// TwinCAT 3 PLC project PLC
// ProgramVersion: 3.1.4026.20
// libraries:
//   Tc2_MC2, * (Beckhoff Automation GmbH)
//   Tc2_Standard, * (Beckhoff Automation GmbH)
//   Tc2_System, * (Beckhoff Automation GmbH)
// project tree:
//   DUTs/ EAnlageGes.TcDUT, EAnlagenStatus.TcDUT, EFoerderband.TcDUT, ETransport.TcDUT
//   GVLs/ IFC_HW.TcGVL
//   / PlcTask.TcTTO
//   POUs/ FB_Abfuellmodul.TcPOU, FB_DigitalInput.TcPOU, FB_Dispenser.TcPOU, MAIN.TcPOU, F_SensStationMonitor.TcPOU
//   POUs/Fehlerbehandlung/ FB_TimeOutError.TcPOU
//   POUs/HardwareEbene/ FB_StatusLight.TcPOU, FB_CNV.TcPOU, FB_RCtrl.TcPOU, FB_Transport.TcPOU
//   POUs/ProzessEbene/ FB_Vereinzelung.TcPOU (not stored)
// (motion and I/O tree: see PLC project tempmodel)
// real-time tasks:
//   TASK PlcTask: cycle T#10ms, priority 21, ADS port 350
//   TASK PlcTask1: cycle T#10ms, priority 22, ADS port 351
//   TASK PlcTask2: cycle T#10ms, priority 20, ADS port 352
// variable links:
//   LF_System_PLC/LF_System_PLC Instance <-> PLC/PLC Instance
//     PlcTask Inputs/MAIN.bIn_LedGreen <-> PlcTask Outputs/IFC_HW.bAmpelGrun
//     PlcTask Inputs/MAIN.bIn_LedRot <-> PlcTask Outputs/IFC_HW.bAmpelRot
//     PlcTask Inputs/MAIN.bIn_LedYellow <-> PlcTask Outputs/IFC_HW.bAmpelGelb
//     PlcTask Inputs/MAIN.bIn_Schleuse1_L1 <-> PlcTask Outputs/IFC_HW.bR1AKT1
//     PlcTask Inputs/MAIN.bIn_Schleuse1_L2 <-> PlcTask Outputs/IFC_HW.bR2AKT1
//     PlcTask Inputs/MAIN.bIn_Schleuse2_L1 <-> PlcTask Outputs/IFC_HW.bR1AKT2
//     PlcTask Inputs/MAIN.bIn_Schleuse2_L2 <-> PlcTask Outputs/IFC_HW.bR2AKT2
//     PlcTask Outputs/MAIN.bEnable <-> PlcTask Inputs/IFC_HW.bEnable
//     PlcTask Outputs/MAIN.bExecute <-> PlcTask Inputs/IFC_HW.bExecute
//     PlcTask Outputs/MAIN.bOut_VereinzelungNS1 <-> PlcTask Inputs/IFC_HW.bEinzelSens3
//     PlcTask Outputs/MAIN.bOut_VereinzelungNS2 <-> PlcTask Inputs/IFC_HW.bEinzelSens2
//     PlcTask Outputs/MAIN.bOut_VereinzelungNS3 <-> PlcTask Inputs/IFC_HW.bEinzelSens1
//   PLC/PLC Instance <-> NC-Task 1 SAF/Axes/BandAchse
//     PlcTask Inputs/IFC_HW.ax_BandMotor.NcToPlc <-> Outputs/ToPlc
//     PlcTask Outputs/IFC_HW.ax_BandMotor.PlcToNc <-> Inputs/FromPlc

CONFIGURATION PLC
    RESOURCE PLC ON TwinCAT3
        TASK PlcTask(INTERVAL := T#10ms, PRIORITY := 20);
        PROGRAM MAIN WITH PlcTask : MAIN;
    END_RESOURCE
END_CONFIGURATION

// ---- DUTs/EAnlageGes.TcDUT
{attribute 'qualified_only'}
{attribute 'strict'}
{attribute 'to_string'}
TYPE EFoerderband :
(
	Off:=0,
	Init := 1,
	Ready := 2,
	Production := 3,
	Done := 4	
);
END_TYPE

// ---- DUTs/EAnlagenStatus.TcDUT
{attribute 'qualified_only'}
{attribute 'strict'}
{attribute 'to_string'}
TYPE EAnlagenStatus:
(
	OFF := 0,
	StateInitOpen := 10,
	StateInitClose := 11,
	StateReady := 20,
	StateProductionOpen := 30,
	StateProductionClose := 31,
	StateDone := 40	
);
END_TYPE

// ---- DUTs/EFoerderband.TcDUT
{attribute 'qualified_only'}
{attribute 'strict'}
{attribute 'to_string'}
TYPE EFoerderband :
(
	Off:=0,
	init := 1,
	ErrorState := 99,
	Resolve := 100,
	Ready := 2,
	CNV_on := 3,
	CNV:aus := 4,
	Done := 5
	
);
END_TYPE

// ---- DUTs/ETransport.TcDUT
{attribute 'qualified_only'}
{attribute 'strict'}
{attribute 'to_string'}
TYPE ETransport :
(
	Off:=0,
	Init := 1,
	Ready := 2,
	Production := 3,
	Producing := 4,
	Done := 5
);
END_TYPE

// ---- GVLs/IFC_HW.TcGVL
// In dieser GVL werden alle Variablen deklariert die auf die realen Klemmen zugreifen
VAR_GLOBAL
	
	// Allgemeine Variablen fur MAIN und HMI
		bEnable		AT%I*	: BOOL;			// Enable Factory (HMI Production Umgebung)
		bExecute	AT%I*	: BOOL;			// Startsignal	(Start Knopf Konsole)
		bStop				: BOOL;			// Stop Variable (interne Variable um FB's zu stoppen)
		bReset				: BOOL;			// Reset Variable
		
	// Station Statusampel	
		bAmpelRot 	AT%Q* 	: BOOL;			// Signal-LED Rot
		bAmpelGelb 	AT%Q* 	: BOOL;			// Signal-LED Gelb
		bAmpelGrun 	AT%Q* 	: BOOL;			// Signal-LED Grun
			
	// Station Vereinzelung
		bEinzelSens1 	AT%I*	: BOOL;					// Separation Sensor 1 (Kammer)
		bEinzelSens2 	AT%I*	: BOOL;					// Separation Sensor 2 (Rohr)
		bEinzelSens3 	AT%I*	: BOOL;					// Separation Sensor 3 (Flasche auf Kopf)
		bR1AKT1 		AT%Q* 	: BOOL := FALSE;		// Relais 1 Aktor 1 (Schleuse Oben öffnen)
		bR2AKT1 		AT%Q* 	: BOOL := TRUE; 		// Relais 2 Aktor 1 (Schleuse Oben schließen)
		bR1AKT2 		AT%Q* 	: BOOL := FALSE;		// Relais 1 Aktor 2 (Schleuse Unten öffne)
		bR2AKT2 		AT%Q* 	: BOOL := TRUE;			// Relais 2 Aktor 2	(Schleuse Unten schließen)
	
	// Station Forderband
		bBandSens1 	AT %I*	: BOOL;		// Forderband Sensor 1 (Extruder 1)
		bBandSens2	AT %I*	: BOOL;		// Forderband Sensor 2 (Extruder 2)
		bBandSens3 	AT %I*	: BOOL;		// Forderband Sensor 3 (Extruder 3)
		bBandSens4 	AT %I*	: BOOL;		// Forderband Sensor 4 (Übergabe Roboter)
		bBandHub1 	AT %Q*	: BOOL;		// Forderband Hubmagnet 1 (Schleuse Extruder 1)
		bBandHub2 	AT %Q*	: BOOL;		// Forderband Hubmagnet 1 (Schleuse Extruder 2)
		bBandHub3 	AT %Q*	: BOOL;		// Forderband Hubmagnet 1 (Schleuse Extruder 3)
		
		ax_Extruder1 	: AXIS_REF;		// Forderband NC-Achse Extruder 1
		ax_Extruder2 	: AXIS_REF;		// Forderband NC-Achse Extruder 2
		ax_Extruder3 	: AXIS_REF;		// Forderband NC-Achse Extruder 3
		ax_BandMotor 	: AXIS_REF;		// Forderband NC-Achse Band
		
		iBandFullmenge1		: INT := 1;	// in Gramm (Soll Füllmenge Extruder 1)
		iBandFullmenge2		: INT := 1;	// in Gramm (Soll Füllmenge Extruder 2)
		iBandFullmenge3		: INT := 1;	// in Gramm (Soll Füllmenge Extruder 3)
		
	//Füllstandsüberwachung
		iFillSens1 AT%I*	: UINT;		// Füllstandssensor im Granulatspeicher 1
		iFillSens2 AT%I*	: UINT;		// Füllstandssensor im Granulatspeicher 2
		iFillSens3 AT%I*	: UINT;		// Füllstandssensor im Granulatspeicher 3
		
		rFillLevelPercent1	: REAL;		// Füllstand im Granulatspeicher 1 in %
		rFillLevelGramm1	: REAL;		// Füllstand im Granulatspeicher 1 in g
		rFillLevelPercent2	: REAL;		// Füllstand im Granulatspeicher 2 in %
		rFillLevelGramm2	: REAL;		// Füllstand im Granulatspeicher 2 in g
		rFillLevelPercent3	: REAL;		// Füllstand im Granulatspeicher 3 in %
		rFillLevelGramm3	: REAL;		// Füllstand im Granulatspeicher 3 in g
		
		rMaxFillLevel 		: REAL := 375;	// Kalibrierter Füllstand für 10% * 10
		
	// Station Waage
		sWaageNachricht		: STRING;	// Nachricht von Wagezelle (fur virtuelle Inbetriebnahme notig)
		bWaageNull			: BOOL;		// TARA Waage (Waage auf Null setzen)
		iWaageMesswert		: INT;		// Messwert der Waage
		
	// Station Behalteridentifikation
		bIdSensorTrager		: BOOL;		// Sensor bei Erkennung eines Datentrager
		sIdNachricht		: STRING;	// Nachricht von RFID-System (fur virtuelle Inbetriebnahme notig)
		sSeriennummer		: STRING;	// Seriennummer RFID-Tag
		
	//Temperierstation
		bVentilator1 	AT %Q*	: BOOL;		// Ventilator 1
		bVentilator2 	AT %Q*	: BOOL;		// Ventilator 2
		bVentilator3 	AT %Q*	: BOOL;		// Ventilator 3
		
		iTempSens1 		AT%I*	: UINT;		// Temperatursensor 1
		iTempSens2 		AT%I*	: UINT;		// Temperatursensor 2
		iHeizpatrone 	AT%Q*	: UINT;		// Heizpatronen
		
		iMaxTemp				: UINT := 5500;		// in °C * 100
		
	// Station Manipulator
		bManEndXmin 		AT%I* 	: BOOL := TRUE;		// Manipulator min Endschalter Achse x
		bManEndYmin 		AT%I* 	: BOOL := TRUE;		// Manipulator min Endschalter Achse y
		bManEndZmin 		AT%I* 	: BOOL := TRUE;		// Manipulator min Endschalter Achse z
		bManEndGmin 		AT%I* 	: BOOL := TRUE;		// Manipulator min Endschalter Achse Gripper
		bManEndXmax 		AT%I* 	: BOOL := TRUE;		// Manipulator max Endschalter Achse x
		bManEndYmax 		AT%I* 	: BOOL := TRUE;		// Manipulator max Endschalter Achse y
		bManEndZmax 		AT%I* 	: BOOL := TRUE;		// Manipulator max Endschalter Achse z
		bManEndGmax 		AT%I* 	: BOOL := TRUE;		// Manipulator max Endschalter Achse Gripper
		bManBrakeZ			AT%Q*	: BOOL := FALSE;	// Bremse Achse z
		
		ax_ManX			: AXIS_REF;			// Manipulator NC-Achse x
		ax_ManY			: AXIS_REF;			// Manipulator NC-Achse y
		ax_ManZ			: AXIS_REF;			// Manipulator NC-Achse z
		ax_ManG			: AXIS_REF; 		// Manipulator NC-Achse Gripper
		
		bGripperClosed		AT%Q*	: BOOL; 			// signal if gripper is closed ONLY USED IN SIM
END_VAR

// ---- POUs/MAIN.TcPOU
PROGRAM MAIN
VAR
	bRed : BOOL;
	bGreen : BOOL;
	bYellow : BOOL;
	
	// FB_Vereinzelung_In:
	bSens1 : BOOL;
	bSens2 : BOOL;
	bSens3 : BOOL;
	bEnable : BOOL;
	bExecute : BOOL;
	
	// FB_Vereinzelung_OUT:
	bGate1 : BOOL;
	bGate2 : BOOL;
	
	fbVereinzelung : FB_Vereinzelung;
	fbRctrl : fb_RCtrl;	
	fbBlink : FB_StatusLight;
	fbCNV : FB_CNV;
	fbEndXmin : FB_DigitalInput(TRUE);
	fbAbfuellmodul : FB_Abfuellmodul;
	
	eStatus : EAnlagenStatus;
	nDoneCounter : INT;
	bError : BOOL;
	ErrorID : DWORD;
	bReset : BOOL;
	
	
	
END_VAR

fbCNV(
	bEnable:= ifc_hw.bEnable, 
	bExecute:= ifc_hw.bExecute, 
	bHalt:= ifc_hw.bBandSens1, 
	rVel:= 50, 
	ax:= ifc_hw.ax_BandMotor);
	
fbEndXmin (bsensSignal := Ifc_HW.bManEndXmin , bSensLogic =>);

IF fbEndXmin.bSensLogic THEN
	//Achse darf nicht in negative Richtung fahren
END_IF
	
fbVereinzelung(
	bSens1 := IFC_HW.bEinzelSens1,
	bSens2 := IFC_HW.bEinzelSens2,
	bSens3 := IFC_HW.bEinzelSens3,
	bEnable := IFC_HW.bEnable,
	bExecute := IFC_HW.bExecute,
	bGate1 => bGate1,
	bGate2 => bGate2,
	eStatus => eStatus,
	nDoneCounter => nDoneCounter);
	
bGate1 := fbVereinzelung.bGate1;
bGate2 := fbVereinzelung.bGate2;

fbRctrl(
	bGate1 := bGate1,
	bGate2 := bGate2,
	bGate1Auf=> IFC_HW.bR1AKT1, 
	bGate1Zu=> IFC_HW.bR2AKT1, 
	bGate2Auf=> IFC_HW.bR1AKT2, 
	bGate2Zu=> IFC_HW.bR2AKT2);

fbAbfuellmodul(
	bEnable:= , 
	bExecute:= , 
	eState=> , 
	bError=> bError, 
	ErrorID=> ErrorID);

fbBlink(eStatus:= eStatus, bRed=> IFC_HW.bAmpelRot, bGreen=> IFC_HW.bAmpelGrun, bYellow=> IFC_HW.bAmpelGelb);

IF bError AND (ErrorID = 9001 OR ErrorID = 9003) THEN
	ifc_HW.bstop := TRUE;
END_IF

ifc_HW.bReset := bReset;
	
IF breset AND NOT bError THEN
	ifc_HW.bStop := FALSE;
	breset := FALSE;
END_IF
(*
//OUT
IFC_HW.bAmpelRot := bRed;
IFC_HW.bAmpelGrun := bGreen;
IFC_HW.bAmpelGelb := bYellow;

IFC_HW.bR1AKT1 := bGate1Auf; //Schleuse oben öffnen
IFC_HW.bR2AKT1 := bGate1Zu;
IFC_HW.bR1AKT2 := bGate2Auf;
IFC_HW.bR2AKT2 := bGate2Zu;

//IN
bSens1 := IFC_HW.bEinzelSens1;
bSens2 := IFC_HW.bEinzelSens1;
bSens3 := IFC_HW.bEinzelSens3;

bEnable := IFC_HW.bEnable;
bExecute := IFC_HW.bExecute;
*)

END_PROGRAM

// ---- POUs/HardwareEbene/FB_RCtrl.TcPOU
FUNCTION_BLOCK FB_RCtrl
VAR_INPUT
	bGate1 : BOOL;
	bGate2 : BOOL;
	
END_VAR
VAR_OUTPUT
	bGate1Auf : BOOL;
	bGate1Zu : BOOL;
	bGate2Auf : BOOL;
	bGate2Zu : BOOL;
END_VAR
VAR
END_VAR

IF bGate1 THEN
	bGate1Auf := TRUE;
	bGate1Zu := FALSE;
	bGate2Auf := FALSE;
	bGate2Zu := TRUE;

ELSIF bGate2 THEN
	bGate1Auf := FALSE;
	bGate1Zu := TRUE;
	bGate2Auf := TRUE;
	bGate2Zu := FALSE;

ELSIF NOT bGate1 THEN
	bGate1Auf := FALSE;
	bGate1Zu := TRUE;

ELSIF NOT bGate2 THEN
	bGate2Auf := FALSE;
	bGate2Zu := TRUE;
	
END_IF

END_FUNCTION_BLOCK

// ---- POUs/HardwareEbene/FB_StatusLight.TcPOU
FUNCTION_BLOCK FB_StatusLight
VAR_INPUT
	eStatus : EAnlagenStatus;
	//bEnable : BOOL; //für stop status
	
END_VAR
VAR_OUTPUT
	bRed : BOOL;
	bGreen : BOOL;
	bYellow : BOOL;
	
END_VAR
VAR
	bblinkEnable : BOOL := FALSE;
	bblinkNow : BOOL := FALSE;
	
	bblinkRED : BOOL := FALSE;
	bblinkGreen : BOOL := FALSE;
	bblinkYellow : BOOL := FALSE;
	
	fbTON : TON;
	fbTP : TP;

END_VAR

bblinkEnable := FALSE;
bblinkNow := FALSE;
	
bblinkRED := FALSE;
bblinkGreen := FALSE;
bblinkYellow := FALSE;

bRed    := FALSE;
bGreen  := FALSE;
bYellow := FALSE;

CASE eStatus OF
	EAnlagenStatus.OFF:
		bRed := TRUE;
		bblinkEnable := FALSE;
		
	EAnlagenStatus.StateInitOpen, EAnlagenStatus.StateInitClose:	//Init
		bblinkEnable := TRUE;
		bblinkGreen := TRUE;
		bblinkRed := FALSE;
		bblinkYellow := FALSE;
		
	EAnlagenStatus.StateProductionOpen, EAnlagenStatus.StateProductionClose: //Production
		bblinkEnable := FALSE;
		bGreen := TRUE;
		
	EAnlagenStatus.StateReady: //Ready
		bblinkEnable := TRUE;
		bblinkGreen := TRUE;
		bblinkyellow := TRUE;
	
	EAnlagenStatus.StateDone: //Done
		bblinkEnable := FALSE;
		bGreen := TRUE;
		bYellow := TRUE;
	
	
END_CASE

fbTON(IN:=bblinkEnable AND NOT fbTon.Q , PT:= T#1S , Q=> , ET=> );
fbTP(IN:= fbTon.Q, PT:= T#500MS , Q=> , ET=> );

bblinkNow := fbTP.Q;

IF bblinkEnable THEN
		
	IF bblinkRed THEN
		bRed := bblinkNow;	
	END_IF
	
	IF bblinkGreen THEN
		bGreen := bblinkNow;
	END_IF
	
	IF bblinkYellow THEN
		bYellow := bblinkNow;
	END_IF
END_IF

END_FUNCTION_BLOCK

// ---- POUs/HardwareEbene/FB_CNV.TcPOU
FUNCTION_BLOCK FB_CNV
VAR_INPUT
	bEnable : BOOL;
	bExecute : BOOL;
	bHalt : BOOL;
	rVel : REAL;
	
	eState : EFoerderband;
END_VAR
VAR_OUTPUT
END_VAR
VAR
	nState : INT :=0;
	mcPower : MC_Power;
	mcReset : MC_Reset;
	mcVelocity : MC_MoveVelocity;
	mcHalt : MC_Halt;
	ErrorID: INT;
	bStop : Bool;
	mcStop: MC_Stop;
END_VAR

VAR_IN_OUT 
	ax : Axis_Ref;
END_VAR

mcHalt(
	Axis:= ax, 
	Execute:= , 
	Deceleration:= , 
	Jerk:= , 
	BufferMode:= , 
	Options:= , 
	Done=> , 
	Busy=> , 
	Active=> , 
	CommandAborted=> , 
	Error=> , 
	ErrorID=> );
	
mcPower(
	Axis:= ax, 
	Enable:= , 
	Enable_Positive:= , 
	Enable_Negative:= , 
	Override:= , 
	BufferMode:= , 
	Options:= , 
	Status=> , 
	Busy=> , 
	Error=> , 
	ErrorID=> );
	
mcReset(
	Axis:= ax, 
	Execute:= , 
	Done=> , 
	Busy=> , 
	Error=> , 
	ErrorID=> );
	
mcVelocity(
	Axis:= ax, 
	Execute:= , 
	Velocity:= rVel, 
	Acceleration:= , 
	Deceleration:= , 
	Jerk:= , 
	Direction:= , 
	BufferMode:= , 
	Options:= , 
	InVelocity=> , 
	Busy=> , 
	Active=> , 
	CommandAborted=> , 
	Error=> , 
	ErrorID=> );

ax.ReadStatus();

bStop := ifc_HW.bStop;
IF bStop THEN
	nState := 80;
END_IF

IF ax.Status.Error THEN 
	nState := 99;
ELSIF NOT bEnable THEN 
	nState := 0;
END_IF

CASE eState OF
	EFoerderband.Off: // OFF
	
		mcReset.Execute := FALSE;
		mcPower.Enable := FALSE;
		mcPower.Enable_Positive := FALSE;
		mcVelocity.Execute := FALSE;
		mcHalt.Execute := FALSE;
		
		
		IF ax.Status.Error THEN 
			nState := 99;
		ELSIF bEnable THEN 
			nState := 1;
		END_IF
	
	EFoerderband.init: //INIT
		
		mcPower.Enable := TRUE;
		mcPower.Enable_Positive := FALSE;
		mcReset.Execute := FALSE;
		mcVelocity.Execute := FALSE;
		mcHalt.Execute := FALSE;
	
		IF mcPower.Status THEN 
			nState :=2;
		END_IF
		
	EFoerderband.Ready: //Ready
		mcPower.Enable := TRUE;
		mcPower.Enable_Positive := FALSE;
		mcReset.Execute := FALSE;
		mcVelocity.Execute := FALSE;
		mcHalt.Execute := FALSE;
		
		IF bExecute THEN 
			nState :=3;
		END_IF
	
	EFoerderband.CNV_on:// CNV an
		mcPower.Enable := TRUE;
		mcPower.Enable_Positive := TRUE;
		mcReset.Execute := FALSE;
		mcVelocity.Execute := TRUE;
		mcHalt.Execute := FALSE;
		
		IF bHalt THEN 
			nState :=4;
		END_IF
	
	EFoerderband.CNV_aus: // CNV aus
		mcPower.Enable := TRUE;
		mcPower.Enable_Positive := TRUE;
		mcReset.Execute := FALSE;
		mcVelocity.Execute := FALSE;
		mcHalt.Execute := TRUE;
		
		IF mcHalt.Done THEN 
			nState :=5;
		END_IF
	
	EFoerderband.Done: // DONE
		mcPower.Enable := TRUE;
		mcPower.Enable_Positive := TRUE;
		mcReset.Execute := FALSE;
		mcVelocity.Execute := FALSE;
		mcHalt.Execute := FALSE;
		
		IF NOT bExecute AND NOT bHalt THEN 
			nState :=2;
		END_IF
	
	EFoerderband.ErrorState: // ERROR 
		mcPower.Enable := FALSE;
		mcPower.Enable_Positive := FALSE;
		mcReset.Execute := FALSE;
		mcVelocity.Execute := FALSE;
		mcHalt.Execute := FALSE;
		
		IF bEnable THEN 
			nState :=100;
		END_IF
	80: //Stop CNV
	mcVelocity.Execute := FALSE;
	mcHalt.Execute := FALSE;
	mcStop.Execute := TRUE;
	
	81: //RE-INIT //noch überarbeiten mit e state und 
	mcVelocity.Execute := FALSE;
	mcHalt.Execute := FALSE;
	mcStop.Execute := FALSE;
	mcReset //auch noch setzen 
	
	
	EFoerderband.Resolve: // Resolve
		mcPower.Enable := TRUE;
		mcPower.Enable_Positive := TRUE;
		mcReset.Execute := FALSE;
		mcVelocity.Execute := FALSE;
		mcHalt.Execute := FALSE;
	
	IF mcReset.Done THEN 
			nState :=1;
		END_IF
END_CASE

END_FUNCTION_BLOCK

// ---- POUs/FB_DigitalInput.TcPOU
FUNCTION_BLOCK FB_DigitalInput
VAR_INPUT
	bSensSignal : BOOL;
END_VAR
VAR_OUTPUT
	bSensLogic : BOOL;
END_VAR
VAR
	_Invert : BOOL := FALSE; //_ damit man weiß ist eine interne variable
END_VAR

IF _Invert THEN
	bSensLogic := NOT bSensSignal;
ELSE
	bSensLogic := bSensSignal;
END_IF

//FB_Init is always available implicitly and it is used primarily for initialization.
//The return value is not evaluated. For a specific influence, you can also declare the
//methods explicitly and provide additional code there with the standard initialization
//code. You can evaluate the return value.
METHOD FB_Init: BOOL
VAR_INPUT
    bInitRetains: BOOL; // TRUE: the retain variables are initialized (reset warm / reset cold)
    bInCopyCode: BOOL;  // TRUE: the instance will be copied to the copy code afterward (online change)   
	Invert : BOOL;
END_VAR
_Invert := Invert;
END_METHOD

END_FUNCTION_BLOCK

// ---- POUs/FB_Abfuellmodul.TcPOU
FUNCTION_BLOCK FB_Abfuellmodul
VAR_INPUT
	bEnable : BOOL;
	bExecute : BOOL;
END_VAR
VAR_OUTPUT
	eState : EAnlageGes;
	bError : BOOL;
	ErrorID : DWORD;
END_VAR
VAR
	fbTransport : FB_Transport;
	fbDispenser : FB_Dispenser;
	nState : INT;
	bStop : BOOL;
END_VAR

fbTransport(
	bSens1:= , 
	bSens2:= , 
	bSens3:= , 
	bSens4:= , 
	bEnabale:= , 
	bExecute:= , 
	nStation:= , 
	eState:= , 
	fSensStationMonitor:= , 
	bHub1=> , 
	bHub2=> , 
	bHub3=> , 
	bError=> bError, 
	ErrorID=> ErrorID);
	
	bStop := ifc_HW.bStop;
	
	IF NOT bEnable THEN
		//noch auszuarbeiten
	END_IF
	
	IF NOT bStop THEN
		CASE nState OF
			//noch auszuarbeiten
		END_CASE
	END_IF

END_FUNCTION_BLOCK

// ---- POUs/HardwareEbene/FB_Transport.TcPOU
FUNCTION_BLOCK FB_Transport
VAR_INPUT
	bSens1 : BOOL;
	bSens2 : BOOL;
	bSens3 : BOOL;
	bSens4 : BOOL;
	bEnabale : BOOL;
	bExecute : BOOL;
	nStation : INT;
	eState : ETransport;
	fSensStationMonitor : F_SensStationMonitor;
	
END_VAR
VAR_OUTPUT
	bHub1 : BOOL;
	bHub2 : BOOL;
	bHub3 : BOOL;
	bError: BOOL;
	ErrorID : DWORD;
END_VAR
VAR
	fbCNV : FB_CNV;
	nState : INT := 0;
	fbTO_Transport : FB_TimeOutError(9001,T#10S);
	bStop : BOOL;
END_VAR

fbCNV(
	bEnable:= , 
	bExecute:= , 
	bHalt:= , 
	rVel:= , 
	eState:= , 
	ax:= );

fbTO_Transport(
	bIN:= eState, 
	bZiel:= , 
	bReset:= , 
	bError=> , 
	ErrorID=> );
	
	
bStop := ifc_HW.bStop;

IF NOT bEnable THEN
	eState := ETransport.Off;
END_IF

CASE eState OF
	
	ETransport.Off:
		fbCNV.bEnable := FALSE;
		fbCNV.bExecute := FALSE;
		fbCNV.bHalt := FALSE;
		bHub1 := FALSE;
		bHub2 := FALSE;
		bHub3 := FALSE;
		
		IF bEnable THEN
			eState := ETransport.Init;
		END_IF
		
	ETransport.Init:
		fbCNV.bEnable := TRUE;
		fbCNV.bExecute := FALSE;
		fbCNV.bHalt := FALSE;
		bHub1 := FALSE;
		bHub2 := FALSE;
		bHub3 := FALSE;
		
		IF NOT (bSens1 AND bSens2 AND bSens3) AND fbCNV.eState = EFoerderband.Ready THEN
			eState := ETransport.Ready;
		END_IF
		
	ETransport.Ready:
		fbCNV.bEnable := TRUE;
		fbCNV.bExecute := FALSE;
		fbCNV.bHalt := FALSE;
		bHub1 := FALSE;
		bHub2 := FALSE;
		bHub3 := FALSE;
		
		IF bExecute THEN
			eState := eTransport.Production;
		END_IF
		
	ETransport.Production:
		fbCNV.bEnable := TRUE;
		fbCNV.bExecute := TRUE;
		fbCNV.bHalt := FALSE;
		bHub1 := FALSE;
		bHub2 := FALSE;
		bHub3 := FALSE;
		
		CASE nStation OF
			1:
				bHub1 := FALSE;
				bHub2 := FALSE;
				bHub3 := FALSE;
			2: 
				bHub1 := TRUE;
				bHub2 := FALSE;
				bHub3 := FALSE;
			3: 
				bHub1 := FALSE;
				bHub2 := TRUE;
				bHub3 := FALSE;
			4:
				bHub1 := FALSE;
				bHub2 := FALSE;
				bHub3 := TRUE;
		END_CASE
	
		IF fSensStationMonitor = TRUE THEN
			eState := ETransport.Producing;
		END_IF
	
	ETransport.Producing:
		fbCNV.bEnable := TRUE;
		fbCNV.bExecute := FALSE;
		fbCNV.bHalt := TRUE;
		bHub1 := FALSE;
		bHub2 := FALSE;
		bHub3 := FALSE;
		
		IF fbCNV.eState = EFoerderband.Done THEN
			eState := ETransport.Done;
		END_IF
	
	ETransport.Done:
		fbCNV.bEnable := TRUE;
		fbCNV.bExecute := FALSE;
		fbCNV.bHalt := FALSE;
		bHub1 := FALSE;
		bHub2 := FALSE;
		bHub3 := FALSE;
		
		IF NOT bExecute THEN
			eState := ETransport.Ready;
		END_IF

END_CASE

END_FUNCTION_BLOCK

// ---- POUs/F_SensStationMonitor.TcPOU
FUNCTION F_SensStationMonitor : BOOL
VAR_INPUT
	bSens1 : BOOL;
	bSens2 : BOOL;
	bSens3 : BOOL;
	
	nStation : INT;
END_VAR
VAR
END_VAR

F_SensStationMonitor := FALSE;

IF bSens1 AND nStation = 1 THEN
	F_SensStationMonitor := TRUE;	
	RETURN;

ELSIF bSens2 AND nStation = 2 THEN
	F_SensStationMonitor := TRUE;
	RETURN;
	
ELSIF bSens3 AND nStation = 3 THEN
	F_SensStationMonitor := TRUE;
	RETURN;
	
ELSE
	F_SensStationMonitor := FALSE;
	RETURN;
	
END_IF

END_FUNCTION

// ---- POUs/Fehlerbehandlung/FB_TimeOutError.TcPOU
FUNCTION_BLOCK FB_TimeOutError
VAR_INPUT
	bIN : BOOL;
	bZiel : BOOL;
	bReset : BOOL;
END_VAR
VAR_OUTPUT
	bError : BOOL;
	ErrorID : DWORD;
END_VAR
VAR
	timer : Ton;
	_ErrorID : DWORD;
	_PT : TIME;
END_VAR

timer(IN:= , PT:= _PT, Q=> , ET=> );

IF bIN THEN
	timer.IN := TRUE;
END_IF

IF bZiel THEN
	timer.IN := FALSE;
END_IF

IF timer.Q THEN
	bError := TRUE;
	ErrorID := _ErrorID;
ELSIF NOT timer.Q OR bReset THEN
	bError := FALSE;
	ErrorID := 0;
END_IF

//FB_Init is always available implicitly and it is used primarily for initialization.
//The return value is not evaluated. For a specific influence, you can also declare the
//methods explicitly and provide additional code there with the standard initialization
//code. You can evaluate the return value.
METHOD FB_Init: BOOL
VAR_INPUT
    bInitRetains: BOOL; // TRUE: the retain variables are initialized (reset warm / reset cold)
    bInCopyCode: BOOL;  // TRUE: the instance will be copied to the copy code afterward (online change)  
	ErrorID : DWORD; 
	PT : TIME;
END_VAR
_ErrorID := ErrorID;

_PT := PT;
END_METHOD

END_FUNCTION_BLOCK

// ---- POUs/FB_Dispenser.TcPOU
FUNCTION_BLOCK FB_Dispenser
VAR_INPUT
	bSens1 : BOOL;
	bSens2 : BOOL;
	bSens3 : BOOL;
	
	bEnable : BOOL;
	bExecute : BOOL;
	
END_VAR
VAR_OUTPUT
	Schnecke1 : BOOL;
	Schnecke2 : BOOL;
	Schnecke3 : BOOL;
END_VAR
VAR
END_VAR

Schnecke1 := FALSE;
Schnecke2 := FALSE;
Schnecke3 := FALSE;

IF bSens1 AND bEnable AND bExecute THEN
	Schnecke1 := TRUE;
	
ELSIF bSens2 AND bEnable AND bExecute THEN
	Schnecke2 := TRUE;
	
ELSIF bSens3 AND bEnable AND bExecute THEN
	Schnecke3 := TRUE;
	
END_IF

END_FUNCTION_BLOCK
